{attribute 'hide'}
VAR_GLOBAL
    nSecret : INT;
END_VAR

(* stored: Version 1.1.0.1
   GVL GVL_Hidden: Id {66666666-6666-6666-6666-666666666602} *)
